// TIA Portal V20 export
DATA_BLOCK "InstShiftCounterOeeDset1"   // DB124
TITLE = Instanz ShiftCounterOeeDset1 / Instance ShiftCounterOeeDset1
{ DB_Accessible_From_OPC_UA := 'FALSE' }
AUTHOR : SICAR
FAMILY : ProdData
// Instanz DB / Instance DB
// stored: DBAccessibleFromOPCUA false, InstanceOfName LSicar_ProdDataShiftCounterOee, InstanceOfType FB
"LSicar_ProdDataShiftCounterOee"
   // VAR_INPUT
   //    numberConfigDataSets { ExternalAccessible := 'False'; ExternalVisible := 'False'; ExternalWritable := 'False'} : Int := 0;
   //    dataSetNumber { ExternalAccessible := 'False'; ExternalVisible := 'False'; ExternalWritable := 'False'} : UInt := 0;
   //    shiftProdTimeTarget { ExternalAccessible := 'False'; ExternalVisible := 'False'; ExternalWritable := 'False'} : Time := T#0MS;
   //    shiftProdTimeExpired { ExternalAccessible := 'False'; ExternalVisible := 'False'; ExternalWritable := 'False'} : Time := T#0MS;
   // END_VAR
   // VAR_IN_OUT
   //    numberOfDataSets : "LSicar_typeNumberOfDataSets";
   //    dataSet : "LSicar_typeShiftCounterOee";
   // END_VAR
   // VAR
   //    statPartsCurrentCount { ExternalAccessible := 'False'; ExternalVisible := 'False'; ExternalWritable := 'False'} : Array[0..10] of "LSicar_typeEdgePulseStruct";
   //    statPartsCurrentCountOk { ExternalAccessible := 'False'; ExternalVisible := 'False'; ExternalWritable := 'False'} : Array[0..10] of "LSicar_typeEdgePulseStruct";
   //    statFactor { ExternalAccessible := 'False'; ExternalVisible := 'False'; ExternalWritable := 'False'} : "LSicar_typeFactorOee";
   //    statTimeFactorTrend { ExternalAccessible := 'False'; ExternalVisible := 'False'; ExternalWritable := 'False'} : Real := 0.0;
   //    statShiftProdTimeTarget { ExternalAccessible := 'False'; ExternalVisible := 'False'; ExternalWritable := 'False'} : Real := 0.0;
   //    statShiftProdTimeExpired { ExternalAccessible := 'False'; ExternalVisible := 'False'; ExternalWritable := 'False'} : Real := 0.0;
   //    statRisEdgeResetAllExt { ExternalAccessible := 'False'; ExternalVisible := 'False'; ExternalWritable := 'False'} : Bool := FALSE;
   //    statPosPulseResetAllExt { ExternalAccessible := 'False'; ExternalVisible := 'False'; ExternalWritable := 'False'} : Bool := FALSE;
   //    statRisEdgeResetAll { ExternalAccessible := 'False'; ExternalVisible := 'False'; ExternalWritable := 'False'} : Bool := FALSE;
   //    statPosPulseResetAll { ExternalAccessible := 'False'; ExternalVisible := 'False'; ExternalWritable := 'False'} : Bool := FALSE;
   // END_VAR
BEGIN
   statPartsCurrentCount[0..10].risEdgeCountUp := FALSE;
   statPartsCurrentCount[0..10].posPulseCountUp := FALSE;
   statPartsCurrentCount[0..10].risEdgeCountDown := FALSE;
   statPartsCurrentCount[0..10].posPulseCountDown := FALSE;
   statPartsCurrentCount[0..10].risEdgeReset := FALSE;
   statPartsCurrentCount[0..10].posPulseReset := FALSE;
   statPartsCurrentCountOk[0..10].risEdgeCountUp := FALSE;
   statPartsCurrentCountOk[0..10].posPulseCountUp := FALSE;
   statPartsCurrentCountOk[0..10].risEdgeCountDown := FALSE;
   statPartsCurrentCountOk[0..10].posPulseCountDown := FALSE;
   statPartsCurrentCountOk[0..10].risEdgeReset := FALSE;
   statPartsCurrentCountOk[0..10].posPulseReset := FALSE;
   statFactor.utilization := 0.0;
   statFactor.efficiency := 0.0;
   statFactor.quality := 0.0;
END_DATA_BLOCK
